{attribute addProperty BoxType "EK1100-0000-0018"}
{attribute addProperty Id "Beckhoff_EP5xxxEK1122Beckhoff_EP5xxxEK1122_5227C47A2096262"}
{attribute addProperty CRC "420084765"}
{attribute addProperty SizeInBites "2096"}
{attribute addProperty SizeInBytes "262"}
TYPE Beckhoff_EP5xxx_1909FC1D EXTENDS EK1100_179A0949 :
STRUCT
	{attribute addProperty Name "Beckhoff_EP5xxxEK1122"}
	Beckhoff_EP5xxxEK1122 : Beckhoff_EP5xxxEK1122_5227C47A;
END_STRUCT
END_TYPE

(* stored: Version 1.2.0.0, ProductVersion 3.1.4024.9
   DUT Beckhoff_EP5xxx_1909FC1D: Id {49199170-1d55-4c01-ac2b-17190cdee48c} *)
